(* PLC project 117_1_V0.5.project, CODESYS CODESYS V3.5 SP17 Patch 3 *)
(* stored: creationDateTime 1970-01-01T00:00:00, modificationDateTime 2026-06-16T22:51:19.9979415 *)

FUNCTION_BLOCK WaitingTimer
  VAR_INPUT
    xExecute : BOOL := FALSE;  (* Включение работы блока *)
    xCondition : BOOL := FALSE;  (* Ожидаемое состояние *)
    tWaitingTime : TIME := TIME#2s0ms;  (* Максимальное время ожидания состояния *)
  END_VAR
  VAR_OUTPUT
    xDone : BOOL;  (* Флаг успешного ожидания состояния *)
    xTimeOutError : BOOL;  (* Флаг ошибки, отсутствие успешного выполнения за заданное время ожидания. *)
  END_VAR
  VAR
    hTask : CmpIecTask.RTS_IEC_HANDLE;  (* Дескриптор (handle) задачи * ) *)
    result : CmpIecTask.RTS_IEC_RESULT;  (* Результат выполнения функций * ) *)
    pCurrentTaskInfo : POINTER TO CmpIecTask.Task_Info2;  (* Указатель на структуру с информацией о задаче * ) *)
    CurrentTaskInfo : CmpIecTask.Task_Info2;  (* Сама структура с данными * ) *)
    intervalTime : TIME;  (* Время цикла в мс *)
    accumulatedTime : TIME;  (* Накопленное время *)
  END_VAR

            // Запись дескриптора текущей задачи в локальную переменную
hTask := CmpIecTask.IecTaskGetCurrent(pResult := ADR(result));

// При успешном получении дискриптора 
IF hTask <> 0 THEN
	// Запрос информации о задаче
    // IecTaskGetInfo3 возвращает указатель на структуру данных о задаче
    pCurrentTaskInfo := CmpIecTask.IecTaskGetInfo3(hIecTask := hTask, pResult := ADR(result));
    // При действительном  указателе, 
    IF pCurrentTaskInfo <> 0 THEN
		// Запись данных в локальную переменную
        CurrentTaskInfo := pCurrentTaskInfo^;
    END_IF 
END_IF

// Записываем полученное время интервала
intervalTime := DWORD_TO_TIME(CurrentTaskInfo.dwInterval / 1000);

//При включении
IF xExecute THEN
	// При отсутвии ошибок
	IF NOT xTimeOutError THEN
		// При наличии требуемого состояния
		IF xCondition AND NOT xTimeOutError THEN 
			// Флаг успешного ожидания
			xDone				:= TRUE;
			// Сброс накопленного времени ожидания
			accumulatedTime		:= T#0MS;
		// При отсутсвии требуемого состояния и отсутствии ошибок
		ELSE
			// Накопление времени ожидания
			accumulatedTime  := accumulatedTime + intervalTime;
			// При достижении максимального времени ожидания
			IF accumulatedTime >= tWaitingTime THEN
				// Флаг ошибки
				xTimeOutError			:= TRUE;
				// Сброс накопленного времени ожидания
				accumulatedTime := T#0MS;
			END_IF
		END_IF
	END_IF
ELSE 
	// Сброс флага успешного ожидания
	xDone				:= FALSE;
	// Сброс флага ошибки
	xTimeOutError		:= FALSE;
	// Сброс накопленного времени ожидания
	accumulatedTime		:= T#0MS;
END_IF

          
END_FUNCTION_BLOCK
